// TIA Portal project "instalacja_cieplna_338a_V15" (V15)

(* hardware
DEVICE "GSD device_1"  GSD.Device.PN
   slot 0: "Rack"  Rail  V1.0
   slot 0: "AL1102_2"  AL1102
   slot 1: "8 Ports_1"  AL1102
DEVICE "GSD device_2"  GSD.Device.PN
   slot 0: "Rack"  Rail  V1.0
   slot 0: "AL1102_3"  AL1102
   slot 1: "8 Ports_1"  AL1102
DEVICE "GSD device_3"  GSD.Device.PN
   slot 0: "Rack"  Rail  V1.0
   slot 0: "AL1102_4"  AL1102
   slot 1: "8 Ports_1"  AL1102
DEVICE "S71500/ET200MP station_2"  S7-1500 station
   slot 0: "Rail_0"  Rack  6ES7 590-1***0-0AA0
   slot 1: "IO device_1"  IM 155-5 PN HF  6ES7 155-5AA00-0AC0  V3.0
   slot 2: "DQ 32x24VDC/0.5A ST_1"  DQ 32x24VDC/0.5A ST  6ES7 522-1BL00-0AB0  V2.0
   slot 3: "AI 8xU/I/RTD/TC ST_1"  AI 8xU/I/RTD/TC ST  6ES7 531-7KF00-0AB0  V2.0
   slot 4: "AQ 4xU/I ST_1"  AQ 4xU/I ST  6ES7 532-5HD00-0AB0  V2.0
DEVICE "S71500/ET200MP station_1"  S7-1500 station
   slot 0: "Rail_0"  Rack  6ES7 590-1***0-0AA0
   slot 1: "PLC_1"  CPU 1513-1 PN  6ES7 513-1AL00-0AB0  V1.1
      slot 3: "CPU display_1"  6ES7591-1XA00-0AA0
*)

// ===== PLC "PLC_1"  CPU 1513-1 PN =====

VAR_GLOBAL   // PLC tag table "Default tag table"
   "Heater_PWR_Out" AT %Q0.3 : Bool;
   "Heater_Tout_In" AT %IW122 : Int;
   "HeatEx_1_Tin_1_In" AT %IW35 : Int;
   "HeatEx_1_Tout_1_In" AT %IW83 : Int;
   "Heater_Flow_In" AT %IW112 : Int;
   "HeatEx_1_Flow_In" AT %IW44 : Int;
   "Heater_Tin_In" AT %IW103 : Int;
   "Heater_Valve_Out" AT %QW8 : Int;
   "HeatEx_1_Valve_Out" AT %QW4 : Int;
   "HeatEx_1_Tin_2_In" AT %IW78 : Int;
   "HeatEx_1_Tout_2_In" AT %IW30 : Int;
   "HeatEx_2_Tin_2_In" AT %IW73 : Int;
   "HeatEx_2_Tin_1_In" AT %IW68 : Int;
   "HeatEx_2_Tout_2_In" AT %IW58 : Int;
   "HeatEx_2_ValveOut" AT %QW6 : Int;
   "HeatEx_2_Flow_In" AT %IW53 : Int;
   "Preassure_In" AT %IW14 : Int;
   "off" AT %M0.0 : Bool;
   "start" AT %M0.1 : Bool;
   "reset" AT %M0.2 : Bool;
   "dist" AT %MD2 : Real;
   "dist_SP" AT %MD6 : Real;
   "test" AT %MD10 : Real;
   "step_dist" AT %MD14 : Real;
   "HeatEx_SP" AT %MD18 : Real;
   "HeatEx_2_Tout1_In" AT %IW98 : Int;
   "Always_OFF" AT %M0.3 : Bool;
   "Preassure_HeatEx_In" AT %IW12 : Int;
   "Preassure_HeatEx_Out" AT %IW18 : Int;
   "Tag_1" AT %QW2 : Int;
   "Tag_2" AT %QW0 : Int;
END_VAR

DATA_BLOCK "Signals_DB"   // DB3
{ S7_Optimized_Access := 'TRUE' }
VERSION : 0.1
   VAR
      PWM_period : Int;
      Heater_PWR : Real;
      Heater_Alarm : Bool;
      Heater_ResetAlarm : Bool;
      Heater_Tin : Real;
      Heater_Tout : Real;
      HeatEx_1_Tin_1 : Real;
      HeatEx_1_Tin_2 : Real;
      HeatEx_1_Tout_1 : Real;
      HeatEx_1_Tout_2 : Real;
      HeatEx_2_Tin_1 : Real;
      HeatEx_2_Tin_2 : Real;
      HeatEx_2_Tout_1 : Real;
      HeatEx_2_Tout_2 : Real;
      Heater_Flow : Real;
      HeatEx_1_Flow : Real;
      HeatEx_2_Flow : Real;
      Heater_Flow_SP : Real;
      Heater_Valve : Real;
      Preassure : Real;
      Preassure_HeatEx_In : Real;
      Preassure_HeatEx_Out : Real;
      HeatEx_1_Flow_SP : Real;
      HeatEx_1_Valve : Real;
      HeatEx_2_FlowSP : Real;
      HeatEx_2_Valve : Real;
   END_VAR
BEGIN
END_DATA_BLOCK

DATA_BLOCK "PWM_DB"   // DB6
{ S7_Optimized_Access := 'TRUE' }
VERSION : 0.1
// stored: InstanceOfName PWM
"PWM"
BEGIN
END_DATA_BLOCK

// folder: System blocks/Program resources

DATA_BLOCK "IEC_Timer_0_DB"   // DB1
{ S7_Optimized_Access := 'TRUE' }
AUTHOR : Simatic
FAMILY : IEC
NAME : IEC_TMR
VERSION : 1.0
// stored: InstanceOfName IEC_TIMER
"IEC_TIMER"
BEGIN
END_DATA_BLOCK

DATA_BLOCK "IEC_Timer_0_DB_1"   // DB2
{ S7_Optimized_Access := 'TRUE' }
AUTHOR : Simatic
FAMILY : IEC
NAME : IEC_TMR
VERSION : 1.0
// stored: InstanceOfName IEC_TIMER
"IEC_TIMER"
BEGIN
END_DATA_BLOCK

DATA_BLOCK "IEC_Timer_0_DB_2"   // DB9
{ S7_Optimized_Access := 'TRUE' }
AUTHOR : Simatic
FAMILY : IEC
NAME : IEC_TMR
VERSION : 1.0
// stored: InstanceOfName IEC_TIMER
"IEC_TIMER"
BEGIN
END_DATA_BLOCK

// folder: (top level)

FUNCTION_BLOCK "PWM"   // FB2, LAD
{ S7_Optimized_Access := 'TRUE' }
VERSION : 0.1
   VAR_INPUT
      width : Int;
      cycle : Int;
   END_VAR
   VAR_IN_OUT
      output : Bool;
   END_VAR
   VAR_TEMP
      T1 : Int;
      T2 : Int;
      czas1 : Time;
      czas2 : Time;
   END_VAR
BEGIN

REGION Network 1
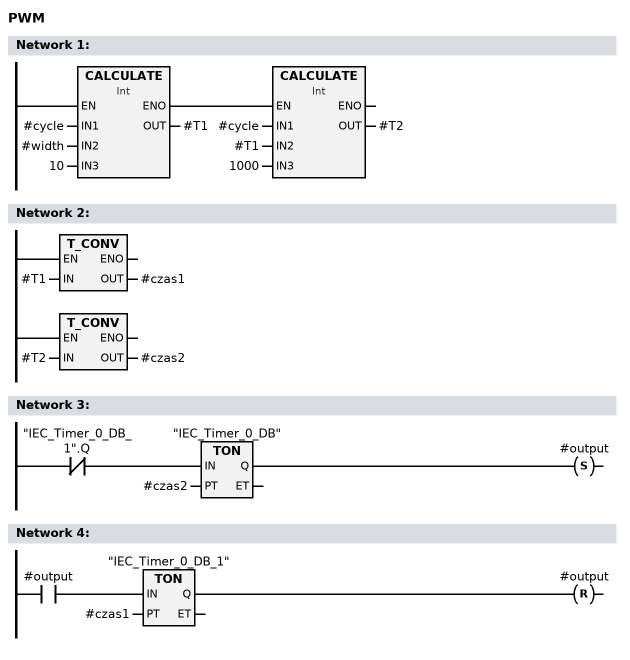
   RUNG wire#powerrail
      { S7_Templates := "SrcType := Int"; S7_GenerateENO := "TRUE"; S7_Expression := "IN1*IN2*IN3" } Calculate(in1 := #cycle, in2 := #width, in3 := 10, out => #T1)
      { S7_Templates := "SrcType := Int"; S7_GenerateENO := "TRUE"; S7_Expression := "IN1*IN3-IN2" } Calculate(in1 := #cycle, in2 := #T1, in3 := 1000, out => #T2)
   END_RUNG
   // the same network as SCL:
   // ENO of a box is taken as its EN; it also drops when the box reports an error
   #T1 := #cycle*#width*10;
   #T2 := #cycle*1000-#T1;
END_REGION

REGION Network 2
   #czas1 := T_CONV(IN := #T1);
   #czas2 := T_CONV(IN := #T2);
END_REGION

REGION Network 3
   "IEC_Timer_0_DB".TON(IN := NOT "IEC_Timer_0_DB_1".Q, PT := #czas2);
   IF "IEC_Timer_0_DB".Q THEN #output := TRUE; END_IF;
END_REGION

REGION Network 4
   "IEC_Timer_0_DB_1".TON(IN := #output, PT := #czas1);
   IF "IEC_Timer_0_DB_1".Q THEN #output := FALSE; END_IF;
END_REGION
END_FUNCTION_BLOCK

ORGANIZATION_BLOCK "Main"   // OB1, LAD, ProgramCycle
TITLE = "Main Program Sweep (Cycle)"
{ S7_Optimized_Access := 'TRUE' }
VERSION : 0.1
   VAR_INPUT
      Initial_Call : Bool;   // Initial call of this OB
      Remanence : Bool;   // =True, if remanent data are available
   END_VAR
   VAR_TEMP
      power_SP_int : Int;
      ret_value : Int;
   END_VAR
BEGIN

REGION Network 1
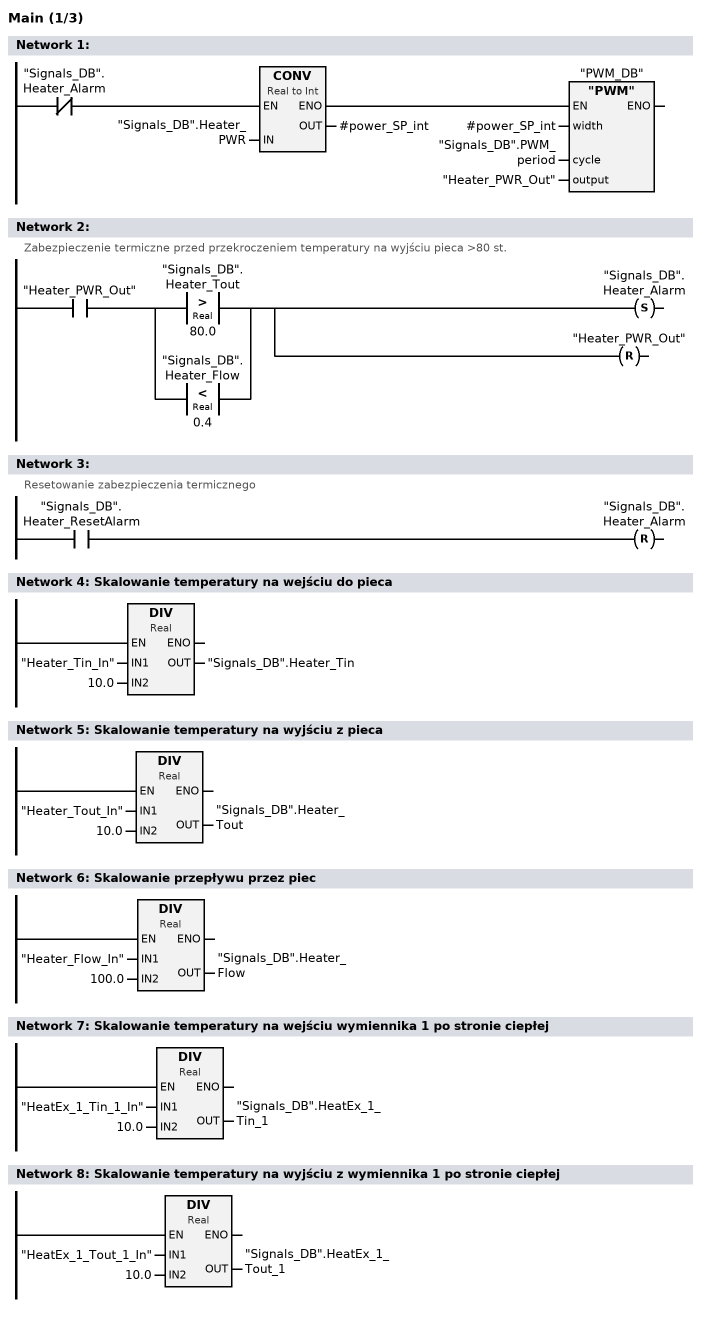
   RUNG wire#powerrail
      I_Contact( "Signals_DB".Heater_Alarm )
      { S7_Templates := "[SrcType := Real, DestType := Int]"; S7_GenerateENO := "TRUE" } Convert(in := "Signals_DB".Heater_PWR, out => #power_SP_int)
      "PWM_DB"(width := #power_SP_int, cycle := "Signals_DB".PWM_period, output := "Heater_PWR_Out")
   END_RUNG
   // the same network as SCL:
   // ENO of a box is taken as its EN; it also drops when the box reports an error
   IF NOT "Signals_DB".Heater_Alarm THEN
       #power_SP_int := REAL_TO_INT("Signals_DB".Heater_PWR);
       "PWM_DB"(width := #power_SP_int, cycle := "Signals_DB".PWM_period, output := "Heater_PWR_Out");   // "PWM"
   END_IF;
END_REGION

REGION Network 2
   // Zabezpieczenie termiczne przed przekroczeniem temperatury na wyjściu pieca >80 st.
   RUNG wire#powerrail
      Contact( "Heater_PWR_Out" )
      wire#w1
      { S7_Templates := "SrcType := Real" } GT_Contact(in1 := "Signals_DB".Heater_Tout, in2 := 80.0)
      wire#w2
      S_Coil( "Signals_DB".Heater_Alarm )
   END_RUNG
   RUNG wire#w1
      { S7_Templates := "SrcType := Real" } LT_Contact(in1 := "Signals_DB".Heater_Flow, in2 := 0.4)
   END_RUNG wire#w2
   RUNG wire#w2
      R_Coil( "Heater_PWR_Out" )
   END_RUNG
   // the same network as SCL:
   IF "Heater_PWR_Out" AND (("Signals_DB".Heater_Tout > 80.0) OR ("Signals_DB".Heater_Flow < 0.4)) THEN
       "Signals_DB".Heater_Alarm := TRUE;
       "Heater_PWR_Out" := FALSE;
   END_IF;
END_REGION

REGION Network 3
   // Resetowanie zabezpieczenia termicznego
   RUNG wire#powerrail
      Contact( "Signals_DB".Heater_ResetAlarm )
      R_Coil( "Signals_DB".Heater_Alarm )
   END_RUNG
   // the same network as SCL:
   IF "Signals_DB".Heater_ResetAlarm THEN "Signals_DB".Heater_Alarm := FALSE; END_IF;
END_REGION

REGION Network 4: Skalowanie temperatury na wejściu do pieca
   RUNG wire#powerrail
      { S7_Templates := "SrcType := Real"; S7_GenerateENO := "TRUE" } Div(in1 := "Heater_Tin_In", in2 := 10.0, out => "Signals_DB".Heater_Tin)
   END_RUNG
   // the same network as SCL:
   "Signals_DB".Heater_Tin := "Heater_Tin_In" / 10.0;
END_REGION

REGION Network 5: Skalowanie temperatury na wyjściu z pieca
   RUNG wire#powerrail
      { S7_Templates := "SrcType := Real"; S7_GenerateENO := "TRUE" } Div(in1 := "Heater_Tout_In", in2 := 10.0, out => "Signals_DB".Heater_Tout)
   END_RUNG
   // the same network as SCL:
   "Signals_DB".Heater_Tout := "Heater_Tout_In" / 10.0;
END_REGION

REGION Network 6: Skalowanie przepływu przez piec
   RUNG wire#powerrail
      { S7_Templates := "SrcType := Real"; S7_GenerateENO := "TRUE" } Div(in1 := "Heater_Flow_In", in2 := 100.0, out => "Signals_DB".Heater_Flow)
   END_RUNG
   // the same network as SCL:
   "Signals_DB".Heater_Flow := "Heater_Flow_In" / 100.0;
END_REGION

REGION Network 7: Skalowanie temperatury na wejściu wymiennika 1 po stronie ciepłej
   RUNG wire#powerrail
      { S7_Templates := "SrcType := Real"; S7_GenerateENO := "TRUE" } Div(in1 := "HeatEx_1_Tin_1_In", in2 := 10.0, out => "Signals_DB".HeatEx_1_Tin_1)
   END_RUNG
   // the same network as SCL:
   "Signals_DB".HeatEx_1_Tin_1 := "HeatEx_1_Tin_1_In" / 10.0;
END_REGION

REGION Network 8: Skalowanie temperatury na wyjściu z wymiennika 1 po stronie ciepłej
   RUNG wire#powerrail
      { S7_Templates := "SrcType := Real"; S7_GenerateENO := "TRUE" } Div(in1 := "HeatEx_1_Tout_1_In", in2 := 10.0, out => "Signals_DB".HeatEx_1_Tout_1)
   END_RUNG
   // the same network as SCL:
   "Signals_DB".HeatEx_1_Tout_1 := "HeatEx_1_Tout_1_In" / 10.0;
END_REGION

REGION Network 9: Skalowanie temperatury na wejściu wymiennika 1 po stronie zimnej
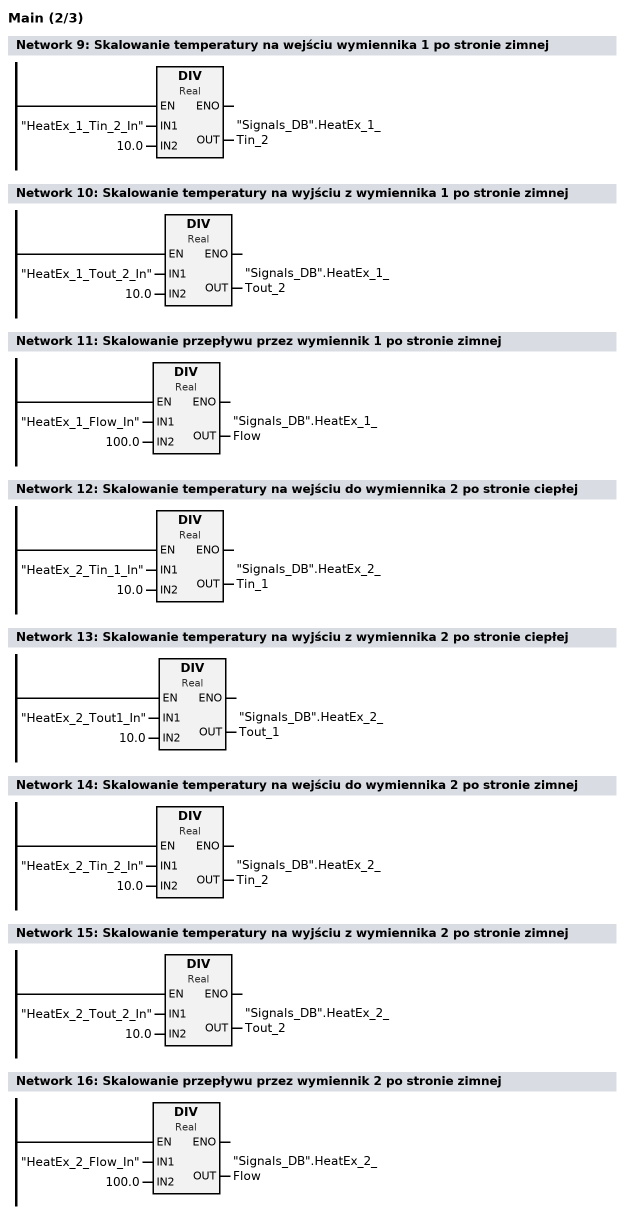
   RUNG wire#powerrail
      { S7_Templates := "SrcType := Real"; S7_GenerateENO := "TRUE" } Div(in1 := "HeatEx_1_Tin_2_In", in2 := 10.0, out => "Signals_DB".HeatEx_1_Tin_2)
   END_RUNG
   // the same network as SCL:
   "Signals_DB".HeatEx_1_Tin_2 := "HeatEx_1_Tin_2_In" / 10.0;
END_REGION

REGION Network 10: Skalowanie temperatury na wyjściu z wymiennika 1 po stronie zimnej
   RUNG wire#powerrail
      { S7_Templates := "SrcType := Real"; S7_GenerateENO := "TRUE" } Div(in1 := "HeatEx_1_Tout_2_In", in2 := 10.0, out => "Signals_DB".HeatEx_1_Tout_2)
   END_RUNG
   // the same network as SCL:
   "Signals_DB".HeatEx_1_Tout_2 := "HeatEx_1_Tout_2_In" / 10.0;
END_REGION

REGION Network 11: Skalowanie przepływu przez wymiennik 1 po stronie zimnej
   RUNG wire#powerrail
      { S7_Templates := "SrcType := Real"; S7_GenerateENO := "TRUE" } Div(in1 := "HeatEx_1_Flow_In", in2 := 100.0, out => "Signals_DB".HeatEx_1_Flow)
   END_RUNG
   // the same network as SCL:
   "Signals_DB".HeatEx_1_Flow := "HeatEx_1_Flow_In" / 100.0;
END_REGION

REGION Network 12: Skalowanie temperatury na wejściu do wymiennika 2 po stronie ciepłej
   RUNG wire#powerrail
      { S7_Templates := "SrcType := Real"; S7_GenerateENO := "TRUE" } Div(in1 := "HeatEx_2_Tin_1_In", in2 := 10.0, out => "Signals_DB".HeatEx_2_Tin_1)
   END_RUNG
   // the same network as SCL:
   "Signals_DB".HeatEx_2_Tin_1 := "HeatEx_2_Tin_1_In" / 10.0;
END_REGION

REGION Network 13: Skalowanie temperatury na wyjściu z wymiennika 2 po stronie ciepłej
   RUNG wire#powerrail
      { S7_Templates := "SrcType := Real"; S7_GenerateENO := "TRUE" } Div(in1 := "HeatEx_2_Tout1_In", in2 := 10.0, out => "Signals_DB".HeatEx_2_Tout_1)
   END_RUNG
   // the same network as SCL:
   "Signals_DB".HeatEx_2_Tout_1 := "HeatEx_2_Tout1_In" / 10.0;
END_REGION

REGION Network 14: Skalowanie temperatury na wejściu do wymiennika 2 po stronie zimnej
   RUNG wire#powerrail
      { S7_Templates := "SrcType := Real"; S7_GenerateENO := "TRUE" } Div(in1 := "HeatEx_2_Tin_2_In", in2 := 10.0, out => "Signals_DB".HeatEx_2_Tin_2)
   END_RUNG
   // the same network as SCL:
   "Signals_DB".HeatEx_2_Tin_2 := "HeatEx_2_Tin_2_In" / 10.0;
END_REGION

REGION Network 15: Skalowanie temperatury na wyjściu z wymiennika 2 po stronie zimnej
   RUNG wire#powerrail
      { S7_Templates := "SrcType := Real"; S7_GenerateENO := "TRUE" } Div(in1 := "HeatEx_2_Tout_2_In", in2 := 10.0, out => "Signals_DB".HeatEx_2_Tout_2)
   END_RUNG
   // the same network as SCL:
   "Signals_DB".HeatEx_2_Tout_2 := "HeatEx_2_Tout_2_In" / 10.0;
END_REGION

REGION Network 16: Skalowanie przepływu przez wymiennik 2 po stronie zimnej
   RUNG wire#powerrail
      { S7_Templates := "SrcType := Real"; S7_GenerateENO := "TRUE" } Div(in1 := "HeatEx_2_Flow_In", in2 := 100.0, out => "Signals_DB".HeatEx_2_Flow)
   END_RUNG
   // the same network as SCL:
   "Signals_DB".HeatEx_2_Flow := "HeatEx_2_Flow_In" / 100.0;
END_REGION

REGION Network 17
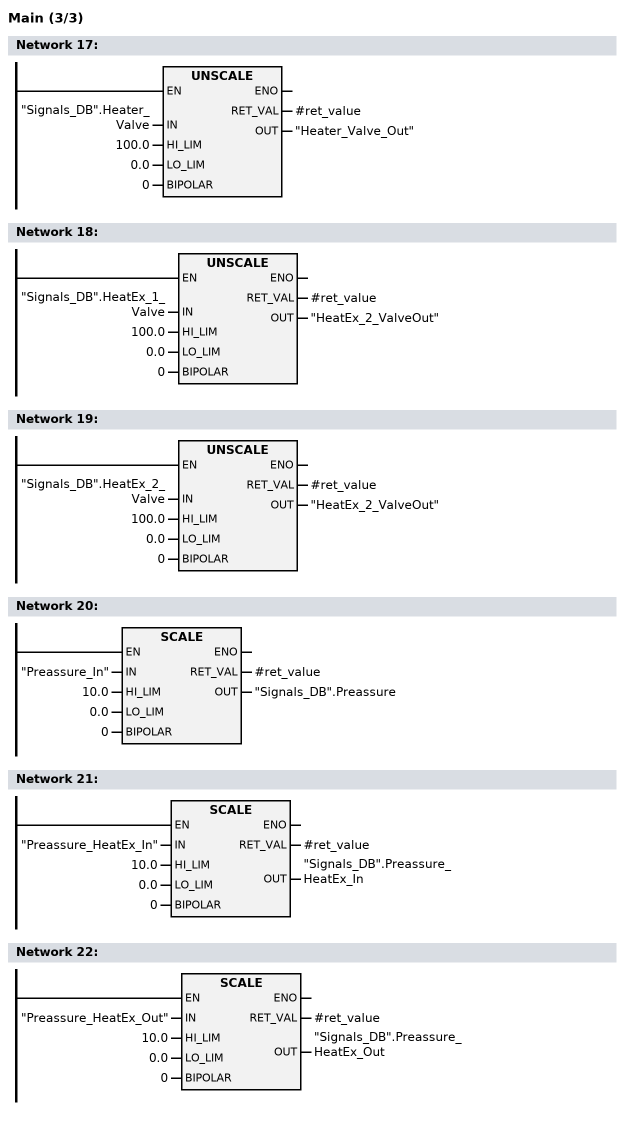
   #ret_value := UNSCALE(IN := "Signals_DB".Heater_Valve,
                         HI_LIM := 100.0,
                         LO_LIM := 0.0,
                         BIPOLAR := 0,
                         OUT => "Heater_Valve_Out");
END_REGION

REGION Network 18
   #ret_value := UNSCALE(IN := "Signals_DB".HeatEx_1_Valve,
                         HI_LIM := 100.0,
                         LO_LIM := 0.0,
                         BIPOLAR := 0,
                         OUT => "HeatEx_2_ValveOut");
END_REGION

REGION Network 19
   #ret_value := UNSCALE(IN := "Signals_DB".HeatEx_2_Valve,
                         HI_LIM := 100.0,
                         LO_LIM := 0.0,
                         BIPOLAR := 0,
                         OUT => "HeatEx_2_ValveOut");
END_REGION

REGION Network 20
   #ret_value := SCALE(IN := "Preassure_In",
                       HI_LIM := 10.0,
                       LO_LIM := 0.0,
                       BIPOLAR := 0,
                       OUT => "Signals_DB".Preassure);
END_REGION

REGION Network 21
   #ret_value := SCALE(IN := "Preassure_HeatEx_In",
                       HI_LIM := 10.0,
                       LO_LIM := 0.0,
                       BIPOLAR := 0,
                       OUT => "Signals_DB".Preassure_HeatEx_In);
END_REGION

REGION Network 22
   #ret_value := SCALE(IN := "Preassure_HeatEx_Out",
                       HI_LIM := 10.0,
                       LO_LIM := 0.0,
                       BIPOLAR := 0,
                       OUT => "Signals_DB".Preassure_HeatEx_Out);
END_REGION
END_ORGANIZATION_BLOCK

ORGANIZATION_BLOCK "Flow controllers"   // OB30, LAD, CyclicInterrupt
{ S7_Optimized_Access := 'TRUE' }
VERSION : 0.1
   VAR_INPUT
      Initial_Call : Bool;   // Initial call of this OB
      Event_Count : Int;   // Events discarded
   END_VAR
BEGIN

REGION Network 1
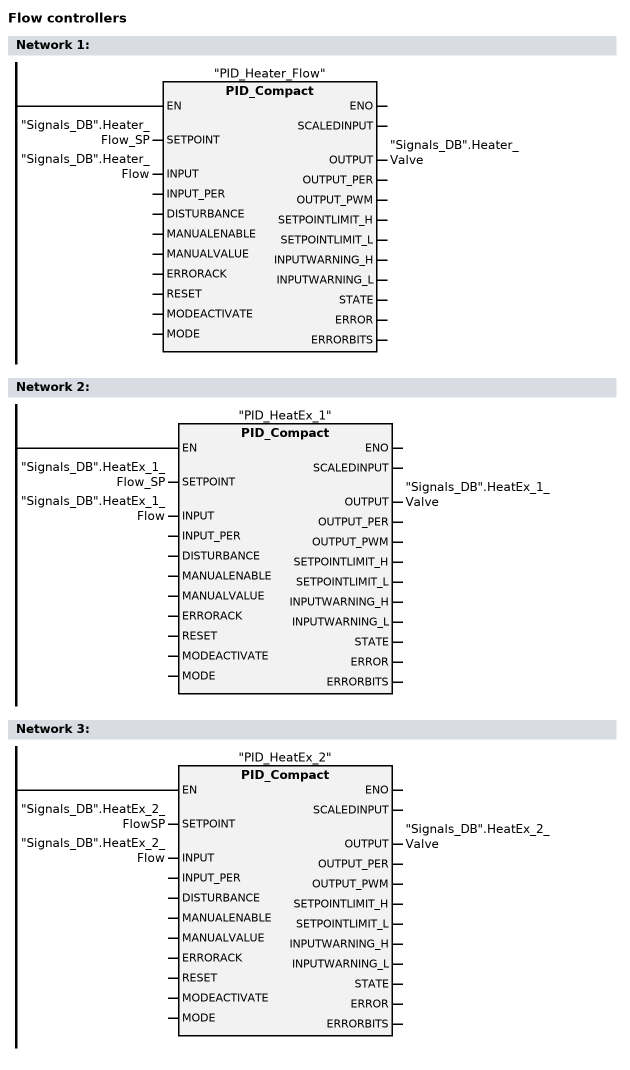
   "PID_Heater_Flow"(Setpoint := "Signals_DB".Heater_Flow_SP,   // PID_Compact
                     Input := "Signals_DB".Heater_Flow,
                     Output => "Signals_DB".Heater_Valve);
END_REGION

REGION Network 2
   "PID_HeatEx_1"(Setpoint := "Signals_DB".HeatEx_1_Flow_SP,   // PID_Compact
                  Input := "Signals_DB".HeatEx_1_Flow,
                  Output => "Signals_DB".HeatEx_1_Valve);
END_REGION

REGION Network 3
   "PID_HeatEx_2"(Setpoint := "Signals_DB".HeatEx_2_FlowSP,   // PID_Compact
                  Input := "Signals_DB".HeatEx_2_Flow,
                  Output => "Signals_DB".HeatEx_2_Valve);
END_REGION
END_ORGANIZATION_BLOCK

ORGANIZATION_BLOCK "Startup"   // OB100, LAD, Startup
TITLE = "Complete Restart"
{ S7_Optimized_Access := 'TRUE' }
VERSION : 0.1
   VAR_INPUT
      LostRetentive : Bool;   // True if retentive data are lost
      LostRTC : Bool;   // True if date and time are lost
   END_VAR
BEGIN

REGION Network 1
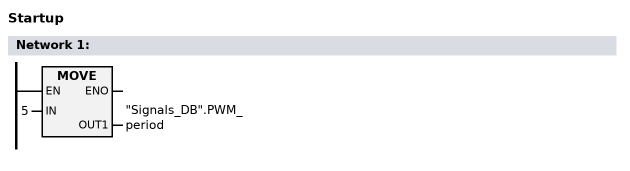
   RUNG wire#powerrail
      { S7_GenerateENO := "TRUE" } Move(in := 5, out1 => "Signals_DB".PWM_period)
   END_RUNG
   // the same network as SCL:
   "Signals_DB".PWM_period := 5;
END_REGION
END_ORGANIZATION_BLOCK